{attribute 'linkalways'} 
{attribute 'no_explicit_call' := 'This FB is a CLASS and must be accessed using methods or properties'}
{attribute 'enable_dynamic_creation'}
FUNCTION_BLOCK Node_ContainerType_Vector_TcVnVector4_INT EXTENDS Node
VAR
    out : _GUID;
END_VAR

METHOD PUBLIC  Clone : I_Node
VAR
	pNode : POINTER TO Node_ContainerType_Vector_TcVnVector4_INT;
END_VAR
pNode := __NEW(Node_ContainerType_Vector_TcVnVector4_INT);
Clone := pNode^;
END_METHOD

METHOD FB_init : BOOL
VAR_INPUT
	bInitRetains : BOOL; // if TRUE, the retain variables are initialized (warm start / cold start)
	bInCopyCode : BOOL;  // if TRUE, the instance afterwards gets moved into the copy code (online change)
END_VAR
AddOutput('out', out);
END_METHOD

METHOD PROTECTED OnExecute
out.Value := ContainerType_Vector_TcVnVector4_INT;
END_METHOD

END_FUNCTION_BLOCK

(* stored: Version 1.1.0.1, ProductVersion 3.1.4026.17
   POU Node_ContainerType_Vector_TcVnVector4_INT: Id {e76b130a-8a4e-0766-02a0-e4b3fbf19da2}, SpecialFunc None
   Folder Constructor: Id {9b70a3d9-130c-0323-27a4-a16215f2fbf1}
   Method Clone: Id {30dc2ab4-cec4-0163-0f29-12b9fb9eb33b}
   Method FB_init: Id {72552922-c541-09d5-0db3-9c71981c54e9}
   Method OnExecute: Id {fab47bee-0ce7-08f8-3cdc-517da795bf86} *)
